INTERFACE I_TakeoverEmulationListener

METHOD M_TakeoverTU_IndexMovedEvent
VAR_INPUT
	mMovedTU_Index	: DINT;
END_VAR
END_METHOD

END_INTERFACE

(* stored: Version 1.1.0.1, ProductVersion 3.1.4022.12
   Itf I_TakeoverEmulationListener: Id {7d920be6-e550-40a3-97d9-38e05e1a47c7}
   Method M_TakeoverTU_IndexMovedEvent: Id {b563a25c-88da-4c31-8117-48cc91f9319f} *)
